TYPE teCTCDeviceStatus :
(
	DEVICE_OK 				:= 0,
	MAINTENANCE_REQUIRED 	:= 1,
	OUT_OF_SPECIFICATION 	:= 2,
	FUNCTIONAL_CHECK 		:= 3,
	FAILURE 				:= 4
);
END_TYPE

(* stored: Version 1.1.0.1, ProductVersion 3.1.4026.17
   EnumerationTextList teCTCDeviceStatus: Id {66465b7e-53bf-4543-86a9-ce618c680989} *)
